FUNCTION_BLOCK F_UPPER_BOUND (* Service Interface Function Block Type *)
  (* Standard: 61131-3; Classification: array function; Description: Copyright (c) 2026 Martin Melik Merkumians This program and the accompanying materials are made available under the terms of the Eclipse Public License 2.0 which is available at https://www.eclipse.org/legal/epl-2.0/ *)
  (* Version 1.0, 2026-03-25, Martin Melik Merkumians *)
  PACKAGE iec61131::arrays;
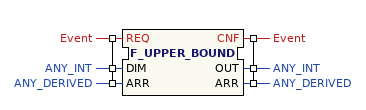
  EVENT_INPUT
    REQ WITH ARR, DIM; (* Service Request *)
  END_EVENT
  EVENT_OUTPUT
    CNF WITH OUT, ARR; (* Confirmation of Requested Service *)
  END_EVENT
  VAR_INPUT
    DIM : ANY_INT := DINT#1; (* Selects array dimension to get the length from, defaults to first dimension *)
  END_VAR
  VAR_OUTPUT
    OUT : ANY_INT; (* Length of the selected array dimension *)
  END_VAR
  VAR_IN_OUT
    ARR : ANY_DERIVED; (* Input array *)
  END_VAR
END_FUNCTION_BLOCK
